// TIA Portal V15.1 export
// export: Created 2024-05-17T05:38:40.4003111Z, ExportSetting WithDefaults, DisplayName Totally Integrated Automation Portal, DisplayVersion V15.1 Update 5, DisplayName TIA Portal Openness, DisplayVersion V15.1 Update 5, DisplayName SINAMICS Startdrive Advanced, DisplayVersion V15.1, DisplayName G130, G150, S120, S150, SINAMICS MV, S210, DisplayVersion V15.1, DisplayName G110M, G120, G120C, G120D, G120P, DisplayVersion V15.1, DisplayName STEP 7 Professional, DisplayVersion V15.1 Update 5, DisplayName STEP 7 Safety, DisplayVersion V15.1, DisplayName WinCC Professional, DisplayVersion V15.1 Update 5, DisplayName SIMATIC Visualization Architect, DisplayVersion V15.1
FUNCTION "LGBDwordTo16Char" : Void   // FC6601, STL
TITLE = convert double-word to 16-numeric-chars
{ S7_Optimized_Access := 'TRUE' }
AUTHOR : Imtech
VERSION : 0.1
// Char 1 ist the lowest
// and
// Char 16 is the highest
// 
// Note
// Char 16 to 11 are always 0
// stored: AutoNumber false, UDAEnableTagReadback false
   VAR_INPUT
      i_dWord : DWord;   // double-word which has to be converted
   END_VAR
   VAR_OUTPUT
      O_cChar1 : Char;   // 1st character of numeric value
      O_cChar2 : Char;   // 2st character of numeric value
      O_cChar3 : Char;   // 3st character of numeric value
      O_cChar4 : Char;   // 4st character of numeric value
      O_cChar5 : Char;   // 5st character of numeric value
      O_cChar6 : Char;   // 6st character of numeric value
      O_cChar7 : Char;   // 7st character of numeric value
      O_cChar8 : Char;   // 8st character of numeric value
      O_cChar9 : Char;   // 9st character of numeric value
      O_cChar10 : Char;   // 10st character of numeric value
      O_cChar11 : Char;   // 11st character of numeric value
      O_cChar12 : Char;   // 12st character of numeric value
      O_cChar13 : Char;   // 13st character of numeric value
      O_cChar14 : Char;   // 14st character of numeric value
      O_cChar15 : Char;   // 15st character of numeric value
      O_cChar16 : Char;   // 16st character of numeric value
   END_VAR
   VAR_TEMP
      tmp_iChar_1 : DInt;
      tmp_iChar_2 : DInt;
      tmp_iChar_3 : DInt;
      tmp_iChar_4 : DInt;
      tmp_iChar_5 : DInt;
      tmp_iChar_6 : DInt;
      tmp_iChar_7 : DInt;
      tmp_iChar_8 : DInt;
      tmp_iChar_9 : DInt;
      tmp_iChar_10 : DInt;
      tmp_iChar_11 : DInt;
      tmp_iChar_12 : DInt;
      tmp_iChar_13 : DInt;
      tmp_iChar_14 : DInt;
      tmp_iChar_15 : DInt;
      tmp_iChar_16 : DInt;
      tmp_i_sum : DInt;
   END_VAR
BEGIN

NETWORK
TITLE = seperat each char of the dword
// Char 10
      L     #i_dWord;
      L     DINT#1000000000;
      /D;
      T     #tmp_iChar_10;

//Char 9
      L     #tmp_iChar_10;
      L     DINT#1000000000;
      *D;
      T     #tmp_i_sum;
      L     #i_dWord;
      L     #tmp_i_sum;
      -D;
      L     DINT#100000000;
      /D;
      T     #tmp_iChar_9;

//Char 8
      L     #tmp_iChar_9;
      L     DINT#100000000;
      *D;
      L     #tmp_i_sum;
      +D;
      T     #tmp_i_sum;
      L     #i_dWord;
      L     #tmp_i_sum;
      -D;
      L     DINT#10000000;
      /D;
      T     #tmp_iChar_8;

//Char 7
      L     #tmp_iChar_8;
      L     DINT#10000000;
      *D;
      L     #tmp_i_sum;
      +D;
      T     #tmp_i_sum;
      L     #i_dWord;
      L     #tmp_i_sum;
      -D;
      L     DINT#1000000;
      /D;
      T     #tmp_iChar_7;

//Char 6
      L     #tmp_iChar_7;
      L     DINT#1000000;
      *D;
      L     #tmp_i_sum;
      +D;
      T     #tmp_i_sum;
      L     #i_dWord;
      L     #tmp_i_sum;
      -D;
      L     DINT#100000;
      /D;
      T     #tmp_iChar_6;

//Char 5
      L     #tmp_iChar_6;
      L     DINT#100000;
      *D;
      L     #tmp_i_sum;
      +D;
      T     #tmp_i_sum;
      L     #i_dWord;
      L     #tmp_i_sum;
      -D;
      L     DINT#10000;
      /D;
      T     #tmp_iChar_5;

//Char 4
      L     #tmp_iChar_5;
      L     DINT#10000;
      *D;
      L     #tmp_i_sum;
      +D;
      T     #tmp_i_sum;
      L     #i_dWord;
      L     #tmp_i_sum;
      -D;
      L     DINT#1000;
      /D;
      T     #tmp_iChar_4;

//Char 3
      L     #tmp_iChar_4;
      L     DINT#1000;
      *D;
      L     #tmp_i_sum;
      +D;
      T     #tmp_i_sum;
      L     #i_dWord;
      L     #tmp_i_sum;
      -D;
      L     DINT#100;
      /D;
      T     #tmp_iChar_3;

//Char 2
      L     #tmp_iChar_3;
      L     DINT#100;
      *D;
      L     #tmp_i_sum;
      +D;
      T     #tmp_i_sum;
      L     #i_dWord;
      L     #tmp_i_sum;
      -D;
      L     DINT#10;
      /D;
      T     #tmp_iChar_2;

//Char 1
      L     #tmp_iChar_2;
      L     DINT#10;
      *D;
      L     #tmp_i_sum;
      +D;
      T     #tmp_i_sum;
      L     #i_dWord;
      L     #tmp_i_sum;
      -D;
      T     #tmp_iChar_1;



NETWORK
TITLE = making out of the int an ASCII
      L     48;
      T     #O_cChar16;

      L     48;
      T     #O_cChar15;

      L     48;
      T     #O_cChar14;

      L     48;
      T     #O_cChar13;

      L     48;
      T     #O_cChar12;

      L     48;
      T     #O_cChar11;

      L     #tmp_iChar_10;
      L     48;
      +I;
      T     #O_cChar10;

      L     #tmp_iChar_9;
      L     48;
      +I;
      T     #O_cChar9;

      L     #tmp_iChar_8;
      L     48;
      +I;
      T     #O_cChar8;

      L     #tmp_iChar_7;
      L     48;
      +I;
      T     #O_cChar7;

      L     #tmp_iChar_6;
      L     48;
      +I;
      T     #O_cChar6;

      L     #tmp_iChar_5;
      L     48;
      +I;
      T     #O_cChar5;

      L     #tmp_iChar_4;
      L     48;
      +I;
      T     #O_cChar4;

      L     #tmp_iChar_3;
      L     48;
      +I;
      T     #O_cChar3;

      L     #tmp_iChar_2;
      L     48;
      +I;
      T     #O_cChar2;

      L     #tmp_iChar_1;
      L     48;
      +I;
      T     #O_cChar1;

      JU    ende;

ende: NOP   0;
END_FUNCTION
